FUNCTION SCODE_CODE : DWORD
VAR_INPUT
	sc		: DWORD;
END_VAR

SCODE_CODE := 16#FFFF AND sc;

END_FUNCTION

(* stored: Version 1.1.0.1, ProductVersion 3.1.4024.12
   POU SCODE_CODE: Id {51f4ad27-9dd2-42d6-b775-99f8a60714ac}, SpecialFunc None *)
